(*
version 1.0	26. oct. 2008
programmer 	hugo
tested by	tobias

This function returns -X

*)
FUNCTION NEGX : REAL
VAR_INPUT
	X : REAL;
END_VAR

NEGX := -X;


(* revision history
hm	26. oct. 2008	rev 1.0
	original version


*)

END_FUNCTION

(* stored: Version 1.1.0.1
   POU NEGX: Id {3b921653-ec23-401e-b1c2-5ca875e924f2}, SpecialFunc None *)
